(*
SPDX-FileCopyrightText: © 2026 Oleksandr Tiutyk <trofimich@gmail.com>
SPDX-License-Identifier: MIT
License: https://opensource.org/license/mit
*)

(*!
<summary>Runs the test automation controller and reports its lifecycle diagnostics.</summary>
<description>
Services the test runner on each TestTask cycle and reports operational state changes and initialization failures.
</description>
*)

PROGRAM MAIN
VAR_OUTPUT
	TestAutomationUnit : TestAutomationController("TestController");
END_VAR
VAR	
	_AutomationControllers : ARRAY [0..0] OF TOF_Automation.IAutomationComponent := 
	[
		TestAutomationUnit
	];
	_StateInitialized : BOOL;
	_LastState : TOF_Automation.OPERATIONAL_STATE;
	_StateMessage : STRING(255);
	_ErrorMessage : TOF_Core.ERROR_MESSAGE;
	_ReasonMessage : STRING(255);
END_VAR
VAR_OUTPUT
	//! <summary>Installed test filter with a task-local diagnostic probe.</summary>
	DiagnosticLogFilter : LogFilter;
	Runner : TOF_Automation.AutomationRunner(components := _AutomationControllers);
END_VAR

IF Runner.State = TOF_Automation.AUTOMATION_RUNNER_STATE.INITIALIZING THEN
	TOF_Core.LogManager.Filter := DiagnosticLogFilter;	
END_IF

Runner.Execute();

IF Runner.State = TOF_Automation.AUTOMATION_RUNNER_STATE.INVALID THEN
	Tc2_System.ADSLOGSTR(
		msgCtrlMask := Tc2_System.Global_Variables.ADSLOG_MSGTYPE_ERROR,
		msgFmtStr := 'CRITICAL: AutomationRunner is INVALID: %s',
		strArg := TO_STRING(Runner.InitializationErrorMessage)
	);
END_IF

IF NOT _StateInitialized OR_ELSE TestAutomationUnit.OperationalState <> _LastState THEN
	_StateInitialized := TRUE;
	_LastState := TestAutomationUnit.OperationalState;
	_StateMessage := TO_STRING(TestAutomationUnit.OperationalState);

	Tc2_System.ADSLOGSTR(
		msgCtrlMask := Tc2_System.Global_Variables.ADSLOG_MSGTYPE_WARN,
		msgFmtStr := 'STATUS: TestAutomationUnit state changed to: %s',
		strArg := _StateMessage
	);

	IF TestAutomationUnit.OperationalState = TOF_Automation.OPERATIONAL_STATE.STOPPED
		OR_ELSE TestAutomationUnit.OperationalState = TOF_Automation.OPERATIONAL_STATE.INVALID
	THEN
		_ReasonMessage := TO_STRING(TestAutomationUnit.OperationalStateReason);
		_ErrorMessage := TestAutomationUnit.Error.TopMessage;

		Tc2_System.ADSLOGSTR(
			msgCtrlMask := Tc2_System.Global_Variables.ADSLOG_MSGTYPE_ERROR,
			msgFmtStr := 'CRITICAL: TestAutomationUnit stopped/failed. Reason: %s',
			strArg := _ReasonMessage
		);

		Tc2_System.ADSLOGSTR(
			msgCtrlMask := Tc2_System.Global_Variables.ADSLOG_MSGTYPE_ERROR,
			msgFmtStr := 'CRITICAL: TestAutomationUnit error message: %s',
			strArg := TO_STRING(_ErrorMessage)
		);
	END_IF
END_IF

END_PROGRAM

(* stored: Version 1.1.0.1, ProductVersion 3.1.4026.20
   POU MAIN: Id {e4eb2eaa-3c4c-0200-2bd5-f94fd2ee20dd}, SpecialFunc None *)
